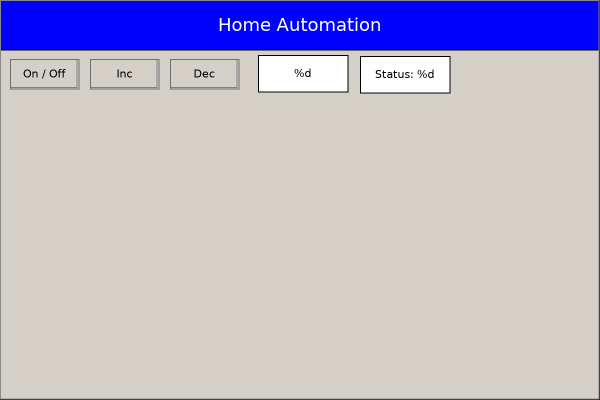
VISUALIZATION V_Main  // 600x400
    Rectangle (0,0 600x400)
    Rectangle (0,0 600x50), "Home Automation"
    Button (10,59 69x30), "On / Off"
        tap PRG_Testing.analogDeviceControl.App_OnOff
    Button (90,59 69x30), "Inc"
        tap PRG_Testing.analogDeviceControl.App_Inc
    Button (170,59 69x30), "Dec"
        tap PRG_Testing.analogDeviceControl.App_Dec
    Rectangle (258,55 90x37), "%d", text variable: PRG_Testing.analogDeviceControl.App_SetValue
        OnMouseClick: write the text variable via VisuDialogs.Numpad, min 0, max 100
    Rectangle (360,56 90x37), "Status: %d", text variable: PRG_Testing.analogStatus
END_VISUALIZATION

(* stored: Version 1.1.0.1, ProductVersion 3.1.4024.13
   Visu V_Main: Id {07ad30e1-4029-4ca7-99be-62a18f71b9f8} *)
